TYPE ST_MixingValveDefaultParameters:
STRUCT
	bFeedbackSignal : BOOL; //true if valve gets a feedback signal for acual position
	fDefaultPosition : REAL; //default position when bSetStatusOn = false
	fControlerAmplification : LREAL;
	fControlerIntegralTime : DINT;
	aSetPointLimitsPosition	: ARRAY[1..2] OF REAL; //setpoint limits for position mode
	aSetPointLimitsTemperature : ARRAY[1..2] OF REAL; //setpoint limits for temperature mode
END_STRUCT
END_TYPE

(* stored: Version 1.1.0.1, ProductVersion 3.1.4024.9
   DUT ST_MixingValveDefaultParameters: Id {fe25e7db-0691-4761-8b7b-8dd172b389e7} *)
